// TIA Portal V18 export
DATA_BLOCK "_screen_home_DB"   // DB75
VERSION : 0.1
// stored: AutoNumber true, DBAccessibleFromOPCUA true, InstanceOfName _screen_Targets, InstanceOfType FB
"_screen_Targets"
   // VAR
   //    t_z : "hmi_home_1";
   //    t_o1 : "hmi_home_1";
   //    t_o2 : "hmi_home_1";
   //    t_x : "hmi_home_1";
   //    t_y : "hmi_home_1";
   //    z : "hmi_home_1";
   //    o1 : "hmi_home_1";
   //    o2 : "hmi_home_1";
   //    x : "hmi_home_1";
   //    y : "hmi_home_1";
   // END_VAR
BEGIN
END_DATA_BLOCK
